// TIA Portal V16 export
// export: Created 2025-08-01T13:38:03.6387301Z, ExportSetting WithDefaults, DisplayName Totally Integrated Automation Portal, DisplayVersion V16, DisplayName TIA Portal Version Control Interface, DisplayVersion V16, DisplayName TIA Portal Openness, DisplayVersion V16, DisplayName STEP 7 Professional, DisplayVersion V16, DisplayName STEP 7 Safety, DisplayVersion V16, DisplayName WinCC Advanced, DisplayVersion V16
DATA_BLOCK "FB_ProductTrigger_1"   // DB67
VERSION : 0.1
// stored: AutoNumber true, InstanceOfName FB_ProductTrigger, InstanceOfType FB
"FB_ProductTrigger"
   // VAR_INPUT
   //    SensorInput : Bool;
   //    TimeDelay : Time;
   //    SystemTime : Time;
   // END_VAR
   // VAR_OUTPUT
   //    TriggerMovement : Bool;
   //    ProductCount : Int;
   // END_VAR
BEGIN
END_DATA_BLOCK
